FUNCTION_BLOCK FB_Test
VAR_INPUT
T	:BOOL;;
END_VAR
VAR_OUTPUT
END_VAR
VAR
END_VAR

T	:=TRUE;
//

END_FUNCTION_BLOCK

(* stored: Version 1.1.0.1, ProductVersion 3.1.4024.3
   POU FB_Test: Id {83ee7ad1-7e96-4758-ada7-f2e2ba9c1f26}, SpecialFunc None *)
